// normalize the input vector
FUNCTION normalize : bool
VAR_IN_OUT
	vec :ARRAY[*] OF LREAL;
END_VAR
VAR
	m,i:DINT;
	vecNorm :LREAL;
END_VAR

m:=UPPER_BOUND(vec,1);
vecNorm :=norm(vec);

// if vector close to zero, remain the same;
IF vecNorm< g_smallNum THEN
	normalize :=FALSE;
	RETURN;
END_IF

FOR i:=1 TO m DO
	vec[i] := vec[i]/vecNorm;
END_FOR

END_FUNCTION

(* stored: Version 1.1.0.1, ProductVersion 3.1.4024.11
   POU normalize: Id {eb641c1c-60d0-4f1d-89d2-38d09d557bbf}, SpecialFunc None *)
